TYPE TcoMessageDigest :
STRUCT
    Digest : DWORD;
    Cycle : ULINT;
    Count : ULINT;
    Category : eMessageCategory;
END_STRUCT
END_TYPE

(* stored: Version 1.1.0.1
   DUT TcoMessageDigest: Id {518a3e34-b85a-0b77-0bb0-128a52748c59} *)
